FUNCTION GetBitFromByte : BOOL
VAR_INPUT
	dataByte : BYTE;
	bitNumber : USINT;
END_VAR
VAR
END_VAR

GetBitFromByte := (SHR(dataByte, bitNumber) AND 1) = 1;

END_FUNCTION

(* stored: Version 1.1.0.1
   POU GetBitFromByte: Id {fae73bce-5cad-0a87-0096-d85ad2ddbe8b}, SpecialFunc None *)
